RoboDK station: delta_robot.rdk

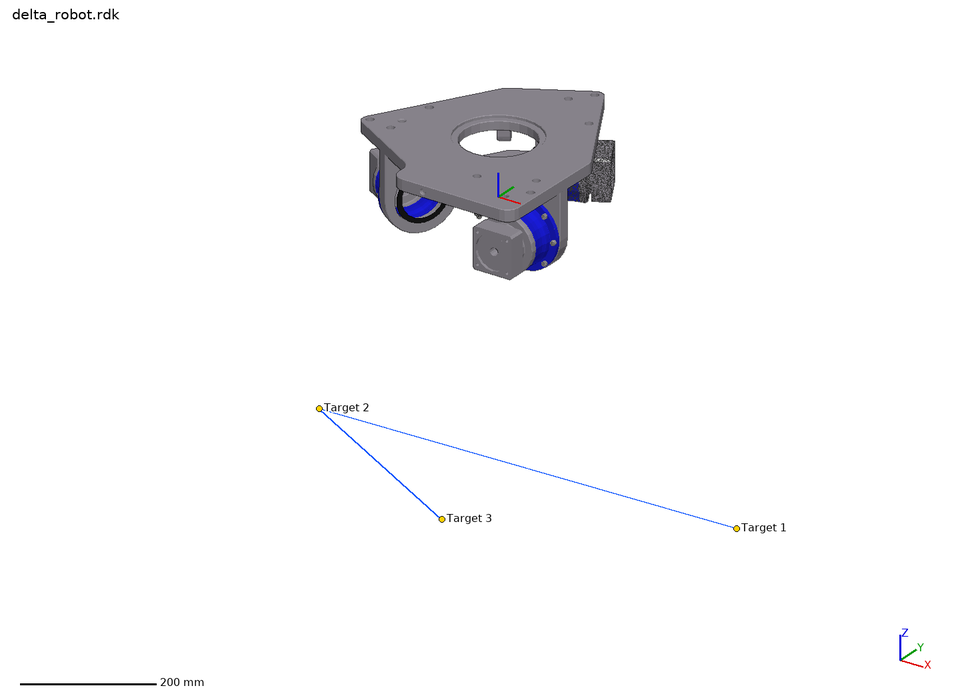
[picture v0: the station drawn from its stored meshes, robots at their saved joint values, targets as dots, program paths as lines]
Station Delta_robot (saved by RoboDK 6.0.6). Poses are relative to the parent item; angles as X-Y-Z fixed-axis rotations.
  - frame autonox Robotics DELTA RL3-600-1kg (A_00072-02) Base at (0, 0, 0) mm
    - robot autonox Robotics DELTA RL3-600-1kg (A_00072-02): 3 axes, payload 1 kg, reach 600 mm, weight 23 kg
        joint limits [-25, -25, -25] to [100, 100, 100]; home [0, 0, 0]; saved at [20.463, 9.913, 13.613]
    - target Target 1 (Cartesian target) at (397.03, 43.43, -448.69) mm, rotated rx 180 ry 0 rz 0 deg; joints [-13.328, 79.53, 73.993] of autonox Robotics DELTA RL3-600-1kg (A_00072-02)
    - target Target 2 (Cartesian target) at (81.11, -575.09, -94) mm, rotated rx 180 ry 0 rz 0 deg; joints [-24.543, -5.987, -22.141] of autonox Robotics DELTA RL3-600-1kg (A_00072-02)
    - target Target 3 (Cartesian target) at (122.95, -320.96, -364.72) mm, rotated rx 180 ry 0 rz 0 deg; joints [0.152, -17.565, 67.48] of autonox Robotics DELTA RL3-600-1kg (A_00072-02)
    - object ASSY GANTRY 5050 at (0, 0, 0) mm, size 50 x 50 x 27.8 mm, geometry from ASSY GANTRY 5050.stp
  - program Prog1 (4 instructions, listed below)
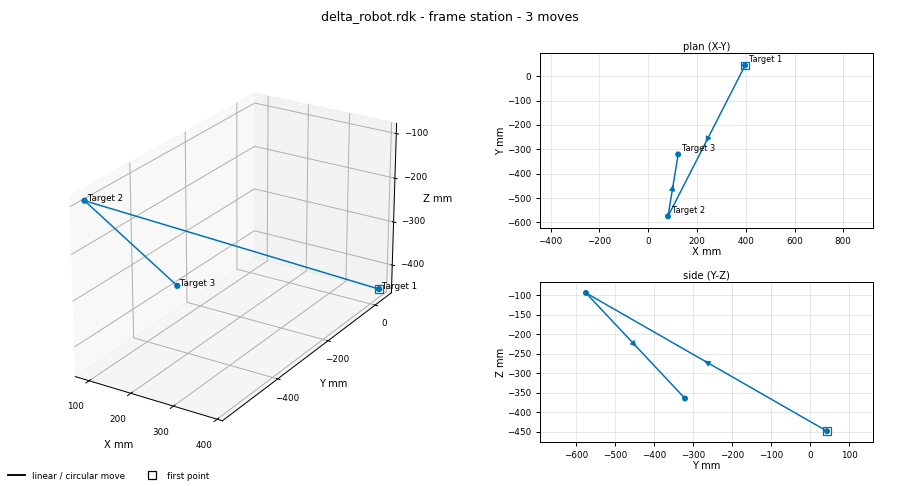
[picture p0: tool path of delta_robot.rdk in frame station, 3 of 3 moves have a stored position in this frame; points joined in program order, loops and branches not executed]

--- program Prog1 (robot autonox Robotics DELTA RL3-600-1kg (A_00072-02)) ---
  Set Ref.: autonox Robotics DELTA RL3-600-1kg (A_00072-02) Base
  MoveJ (Target 1)
  MoveL (Target 2)
  MoveL (Target 3)
